// TIA Portal V19 export
FUNCTION_BLOCK "TYPIC_C301_BF_VEN"   // FB2, FBD
TITLE = TYPIC_C301_BF_VEN: Ventilatie verkeerskoker
{ S7_Optimized_Access := 'TRUE' }
AUTHOR : OCOTECH
FAMILY : Typical
NAME : C301.801
// Logisch Object Besturing: C301.801
// 
// Het doel van de BF ventilatie is de algemene opvolging, sturing en bediening van de ventilatie van een verkeerskoker.
// stored: MemoryReserve 10, SetENOAutomatically false
   VAR_INPUT
      CFG_TST_UTYD { ExternalAccessible := 'False'; ExternalVisible := 'False'; ExternalWritable := 'False'} : Time;   // Maximale transitietijd stand verandering ventilatie (transitiestatus niet bereikt)
      CFG_TST_OK_TYD { ExternalAccessible := 'False'; ExternalVisible := 'False'; ExternalWritable := 'False'} : Time;   // Stabilisatietijd voor de toestand OK (bereikt)
      CFG_ONHD_TYD { ExternalAccessible := 'False'; ExternalVisible := 'False'; ExternalWritable := 'False'} : Time;   // Waarschuwingstijd start automatische onderhoudstesten
      CFG_MAX_NOK1 { ExternalAccessible := 'False'; ExternalVisible := 'False'; ExternalWritable := 'False'} : Int;   // Maximum aantal onbestuurbare ventilatoren voor beschikbaarheidsstatus beschikbaar
      CFG_MAX_NOK2 { ExternalAccessible := 'False'; ExternalVisible := 'False'; ExternalWritable := 'False'} : Int;   // Maximum aantal onbestuurbare ventilatoren voor beschikbaarheidsstatus beperkt beschikbaar
      STU_CMD_AUT { ExternalAccessible := 'False'; ExternalVisible := 'False'; ExternalWritable := 'False'} : USInt;   // Groepscommando: schakel in automatisch
      STU_AUT_CMD { ExternalAccessible := 'False'; ExternalVisible := 'False'; ExternalWritable := 'False'} : USInt;   // Sturing ventilatie algemeen
      STU_AUT_CMD_DIR { ExternalAccessible := 'False'; ExternalVisible := 'False'; ExternalWritable := 'False'} : USInt;   // Sturing richting
      STU_AUT_VGV_BEV { ExternalAccessible := 'False'; ExternalVisible := 'False'; ExternalWritable := 'False'} : USInt;   // Vrijgave ventilator-beveiligingen onbalans en temperatuur
      STU_VGV_ONHD { ExternalAccessible := 'False'; ExternalVisible := 'False'; ExternalWritable := 'False'} : USInt;   // Vrijgave uitvoeren automatische onderhoudstesten
      STU_ALG_LCK_SIG { ExternalAccessible := 'False'; ExternalVisible := 'False'; ExternalWritable := 'False'} : USInt;   // Onderdruk alarmen
      STU_REG_CAPA { ExternalAccessible := 'False'; ExternalVisible := 'False'; ExternalWritable := 'False'} : USInt;   // Gewenste stand ventilatie bij sensorregeling (afkomstig van CF zichthandhaving)
      STU_ENE_VGV_AAN { ExternalAccessible := 'False'; ExternalVisible := 'False'; ExternalWritable := 'False'} : USInt;   // Vrijgeven of verhinderen bijschakelen energieverbruikers (verlichting / ventilatie)
      STU_ENE_MAX_AAN { ExternalAccessible := 'False'; ExternalVisible := 'False'; ExternalWritable := 'False'} : USInt;   // Maximaal toegelaten ventilatiestand
   END_VAR
   VAR_OUTPUT
      STU_CLUST { ExternalAccessible := 'False'; ExternalVisible := 'False'; ExternalWritable := 'False'} : "C301_STU_CLUST_TYPIC";   // Groepscommando met sturingen naar alle clusters van de ventilatiezone
      VAR_PWR { ExternalAccessible := 'False'; ExternalVisible := 'False'; ExternalWritable := 'False'} : Real;   // Som actueel vermogen van alle clusters
      VAR_CAPA { ExternalAccessible := 'False'; ExternalVisible := 'False'; ExternalWritable := 'False'} : USInt;   // De ingestelde ventilatiestand
      VAR_DIR { ExternalAccessible := 'False'; ExternalVisible := 'False'; ExternalWritable := 'False'} : USInt;   // De ingestelde ventilatierichting
   END_VAR
   VAR_IN_OUT
      CFG_CAPA_DIR1 : Array[1..8] of USInt;   // Omzetting ventilatiestand naar aantal ventilatoren, per cluster (zie verder), rijrichting
      CFG_CAPA_DIR2 : Array[1..8] of USInt;   // Omzetting ventilatiestand naar aantal ventilatoren, per cluster (zie verder), tegenrijrichting
      VAR_CLUST : Array[*] of "C301_VAR_CLUST_TYPIC";   // Array met alle clusters, met alle variabelen van de cluster
   END_VAR
   VAR
      BED : Struct   // Bedieningen
         ALG : Struct   // Gewenste stand
            X : "UDT_BED_ALG";
            KNOP { S7_SetPoint := 'True'} : Array[0..10] of "UDT_BED_KNOP";
         END_STRUCT;
         ALG_DIR : Struct   // Gewenste richting
            X : "UDT_BED_ALG";
            KNOP { S7_SetPoint := 'True'} : Array[0..2] of "UDT_BED_KNOP";
         END_STRUCT;
         VGV_BEV : Struct   // Vrijgave ventilator-beveiligingen onbalans en temperatuur
            X : "UDT_BED_ALG";
            KNOP { S7_SetPoint := 'True'} : Array[0..2] of "UDT_BED_KNOP";
         END_STRUCT;
         ONHD : Struct   // Uitvoeren automatische onderhoudstesten
            X : "UDT_BED_ALG";
            KNOP { S7_SetPoint := 'True'} : Array[0..1] of "UDT_BED_KNOP";
         END_STRUCT;
      END_STRUCT;
      BED_ALG { ExternalWritable := 'False'} : "TYPIC_HF_BED_ALG_KNOP";   // Gewenste stand
      BED_ALG_DIR { ExternalWritable := 'False'} : "TYPIC_HF_BED_ALG_KNOP";   // Gewenste richting
      BED_VGV_BEV { ExternalWritable := 'False'} : "TYPIC_HF_BED_ALG_KNOP";   // Vrijgave ventilator-beveiligingen onbalans en temperatuur
      BED_ONHD { ExternalWritable := 'False'} : "TYPIC_HF_BED_ALG_KNOP";   // Uitvoeren automatische onderhoudstesten
      SIG { ExternalWritable := 'False'} : Struct   // Signaleringen
         AA01 : Bool;   // Gewenste stand niet bereikt
         AA02 : Bool;   // Automatische onderhoudstesten ventilatie
         AB01 : Bool;   // Ventilatie niet beschikbaar
         AB02 : Bool;   // Ventilatie beperkt beschikbaar
      END_STRUCT;
      VAR { ExternalWritable := 'False'} : Struct   // Variabelen
         AUT_SWA : USInt;   // De stand die de ventilatie moet handhaven als de bedieningswijze is ingesteld op automatisch
         REG_CAPA : USInt;   // De stand die de ventilatie moet handhaven als de sensorregeling actief is. Deze waarde wordt bepaald door de coordinerende functie Zichthandhaving Verkeerskoker
         BMO : USInt;   // Bedieningsmode
         AUT_DIR : USInt;   // De richting die de ventilatoren op moeten blazen als de bedieningswijze is ingesteld op automatisch
         DIR_BWA : USInt;   // De werkelijke ventilatierichting
         NIV_BWA : USInt;   // Momentane ventilatieniveau (percentage)
         NIV_AAN_BWA { ExternalAccessible := 'False'; ExternalVisible := 'False'} : USInt;   // Momentaan aantal aangeschakelde ventilatoren
         NIV_AAN_SWA { ExternalAccessible := 'False'; ExternalVisible := 'False'} : USInt;   // Gewenst aantal aangeschakelde ventilatoren
         CAPA_MAX { ExternalAccessible := 'False'; ExternalVisible := 'False'} : USInt;   // Totaal aantal ventilatoren in de ventilatiezone
         CAPA_OK_BWA { ExternalAccessible := 'False'; ExternalVisible := 'False'} : USInt;   // Aantal beschikbare ventilatoren
         CAPA_BWA : USInt;   // De totaal beschikbare ventilatiecapaciteit.
         TST_BWA : USInt;   // De status van de transitie van de langsventilatie
         BSC : USInt;   // Geeft de beschikbaarheid van de langsventilatie aan
         VGV_SIG_VOP : USInt;   // TRUE = Signaleringen vrijgegeven voor verkeersoperator FALSE = Onderdrukt
         ONHD_STS : USInt;   // Status automatische onderhoudstesten
         ONHD_CLUST : USInt;   // Nummer van de cluster die onderhoudstesten dient uit te voeren
         VGV_BEV : USInt;   // Vrijgave ventilator-beveiligingen onbalans en temperatuur
         CAPA : USInt;   // De ingestelde ventilatiestand
         DIR : USInt;   // De ingestelde ventilatierichting
      END_STRUCT;
      HF_TST { ExternalAccessible := 'False'; ExternalVisible := 'False'; ExternalWritable := 'False'} : "TYPIC_HF_TST";   // Hulpfunctie transitiestatus
   END_VAR
   // // BED.ALG.KNOP[0] : Auto
   // // BED.ALG.KNOP[1] : 0 (Uit)
   // // BED.ALG.KNOP[2] : 1
   // // BED.ALG.KNOP[3] : 2
   // // BED.ALG.KNOP[4] : 3
   // // BED.ALG.KNOP[5] : 4
   // // BED.ALG.KNOP[6] : 5
   // // BED.ALG.KNOP[7] : 6
   // // BED.ALG.KNOP[8] : 7
   // // BED.ALG.KNOP[9] : 8
   // // BED.ALG.KNOP[10] : Sensorregeling
   // // BED.ALG_DIR.KNOP[0] : Auto
   // // BED.ALG_DIR.KNOP[1] : Rijrichting
   // // BED.ALG_DIR.KNOP[2] : Tegenrij
   // // BED.VGV_BEV.KNOP[0] : Auto
   // // BED.VGV_BEV.KNOP[1] : Ja
   // // BED.VGV_BEV.KNOP[2] : Onderdrukt
   // // BED.ONHD.KNOP[0] : Aan
   // // BED.ONHD.KNOP[1] : Uit
BEGIN

REGION Network 1: START
END_REGION

REGION Network 2: +++ Bedieningen +++
   // Vrijgave en verwerking van de bedieningen (centrale en lokale bediening). De bedienwaardes worden daarna in de verdere deelfunctionaliteiten gebruikt.
END_REGION

REGION Network 3: Knoppen BED_ALG(Gewenste stand)
   // Waardes en vrijge van de knoppen BED_ALG
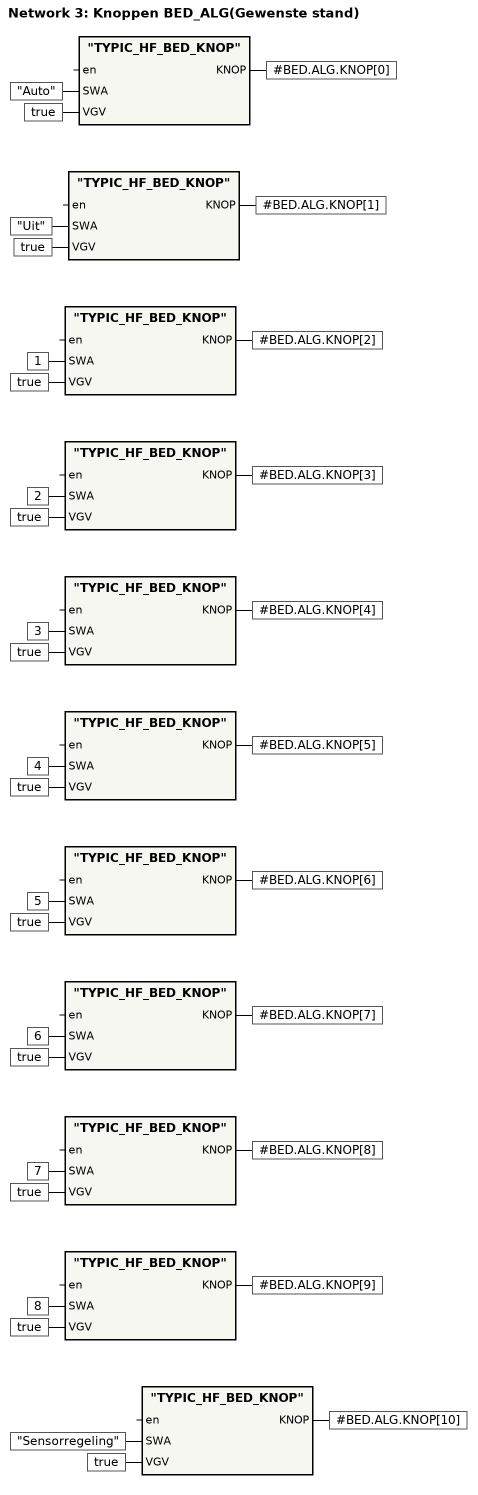
   "TYPIC_HF_BED_KNOP"(SWA := "Auto", VGV := true, KNOP => #BED.ALG.KNOP[0]);
   "TYPIC_HF_BED_KNOP"(SWA := "Uit", VGV := true, KNOP => #BED.ALG.KNOP[1]);
   "TYPIC_HF_BED_KNOP"(SWA := 1, VGV := true, KNOP => #BED.ALG.KNOP[2]);
   "TYPIC_HF_BED_KNOP"(SWA := 2, VGV := true, KNOP => #BED.ALG.KNOP[3]);
   "TYPIC_HF_BED_KNOP"(SWA := 3, VGV := true, KNOP => #BED.ALG.KNOP[4]);
   "TYPIC_HF_BED_KNOP"(SWA := 4, VGV := true, KNOP => #BED.ALG.KNOP[5]);
   "TYPIC_HF_BED_KNOP"(SWA := 5, VGV := true, KNOP => #BED.ALG.KNOP[6]);
   "TYPIC_HF_BED_KNOP"(SWA := 6, VGV := true, KNOP => #BED.ALG.KNOP[7]);
   "TYPIC_HF_BED_KNOP"(SWA := 7, VGV := true, KNOP => #BED.ALG.KNOP[8]);
   "TYPIC_HF_BED_KNOP"(SWA := 8, VGV := true, KNOP => #BED.ALG.KNOP[9]);
   "TYPIC_HF_BED_KNOP"(SWA := "Sensorregeling", VGV := true, KNOP => #BED.ALG.KNOP[10]);
END_REGION

REGION Network 4: BED_ALG(Gewenste stand)
   // Verwerking BED_ALG
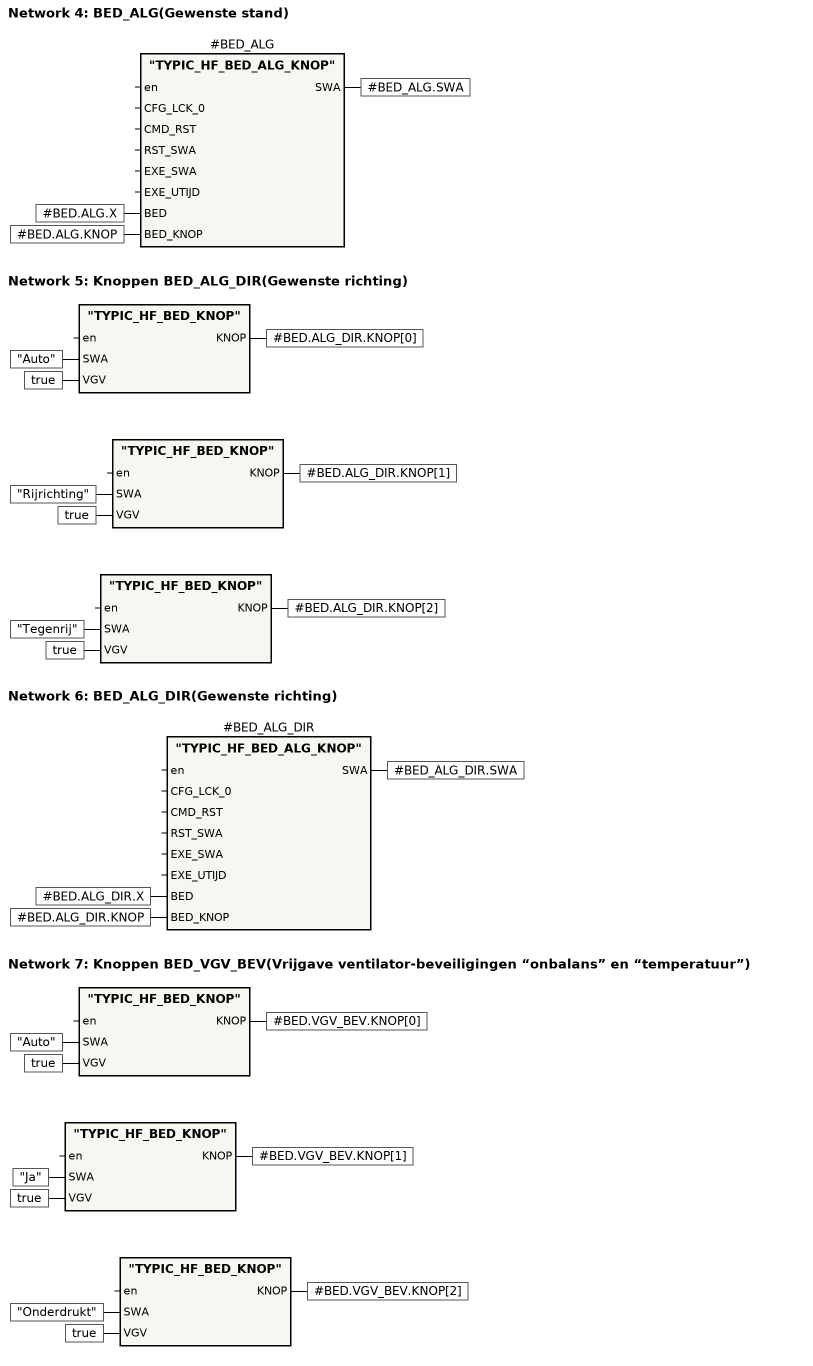
   #BED_ALG(BED := #BED.ALG.X, BED_KNOP := #BED.ALG.KNOP, SWA => #BED_ALG.SWA);   // "TYPIC_HF_BED_ALG_KNOP"
END_REGION

REGION Network 5: Knoppen BED_ALG_DIR(Gewenste richting)
   // Waardes en vrijge van de knoppen BED_ALG_DIR
   "TYPIC_HF_BED_KNOP"(SWA := "Auto", VGV := true, KNOP => #BED.ALG_DIR.KNOP[0]);
   "TYPIC_HF_BED_KNOP"(SWA := "Rijrichting", VGV := true, KNOP => #BED.ALG_DIR.KNOP[1]);
   "TYPIC_HF_BED_KNOP"(SWA := "Tegenrij", VGV := true, KNOP => #BED.ALG_DIR.KNOP[2]);
END_REGION

REGION Network 6: BED_ALG_DIR(Gewenste richting)
   // Verwerking BED_ALG_DIR
   #BED_ALG_DIR(BED := #BED.ALG_DIR.X, BED_KNOP := #BED.ALG_DIR.KNOP, SWA => #BED_ALG_DIR.SWA);   // "TYPIC_HF_BED_ALG_KNOP"
END_REGION

REGION Network 7: Knoppen BED_VGV_BEV(Vrijgave ventilator-beveiligingen “onbalans” en “temperatuur”)
   // Waardes en vrijge van de knoppen BED_VGV_BEV
   "TYPIC_HF_BED_KNOP"(SWA := "Auto", VGV := true, KNOP => #BED.VGV_BEV.KNOP[0]);
   "TYPIC_HF_BED_KNOP"(SWA := "Ja", VGV := true, KNOP => #BED.VGV_BEV.KNOP[1]);
   "TYPIC_HF_BED_KNOP"(SWA := "Onderdrukt", VGV := true, KNOP => #BED.VGV_BEV.KNOP[2]);
END_REGION

REGION Network 8: BED_VGV_BEV(Vrijgave ventilator-beveiligingen “onbalans” en “temperatuur”)
   // Verwerking BED_VGV_BEV
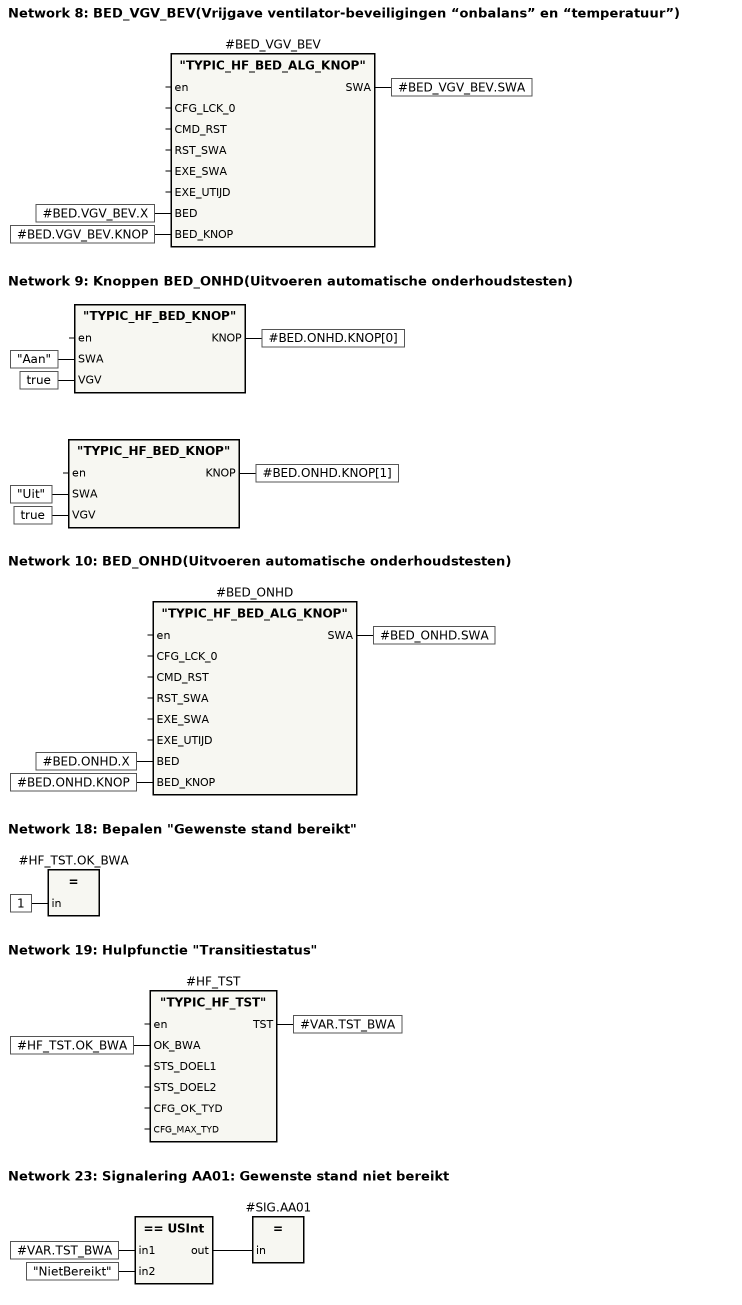
   #BED_VGV_BEV(BED := #BED.VGV_BEV.X, BED_KNOP := #BED.VGV_BEV.KNOP, SWA => #BED_VGV_BEV.SWA);   // "TYPIC_HF_BED_ALG_KNOP"
END_REGION

REGION Network 9: Knoppen BED_ONHD(Uitvoeren automatische onderhoudstesten)
   // Waardes en vrijge van de knoppen BED_ONHD
   "TYPIC_HF_BED_KNOP"(SWA := "Aan", VGV := true, KNOP => #BED.ONHD.KNOP[0]);
   "TYPIC_HF_BED_KNOP"(SWA := "Uit", VGV := true, KNOP => #BED.ONHD.KNOP[1]);
END_REGION

REGION Network 10: BED_ONHD(Uitvoeren automatische onderhoudstesten)
   // Verwerking BED_ONHD
   #BED_ONHD(BED := #BED.ONHD.X, BED_KNOP := #BED.ONHD.KNOP, SWA => #BED_ONHD.SWA);   // "TYPIC_HF_BED_ALG_KNOP"
END_REGION

REGION Network 11: +++ Bepalen bedieningsmode +++
   // Bedieningsmode (Auto / Manueel ) bepalen.
END_REGION

REGION Network 12: +++ Bepalen gewenste capaciteitsinstelling +++
   // Bepalen van de gewenste stand (0..8).
END_REGION

REGION Network 13: +++ Bepalen gewenste ventilatierichting +++
   // Bepalen van de gewenste draairichting (Rijrichting / Tegenrij).
END_REGION

REGION Network 14: +++ Bepalen vrijgave ventilatorbeveiligingen +++
   // Bepalen vrijgave of onderdrukken van de ventilatorbeveiligingen onbalans en temperatuur.
END_REGION

REGION Network 15: +++ Bepalen werkelijke ventilatierichting +++
   // Bepalen van de werkelijke ventilatierichting (Rijrichting / Tegenrij / Onbepaald) aan de hand van de ventilatierichtingen van de ventilatieclusters.
END_REGION

REGION Network 16: +++ Berekeningen +++
   // Verscheidene berekeningen die nodig zijn voor de functionele werking of info voor weergave via de centrale en lokale bediening, zoals het momentane ventilatieniveau, aantal beschikbare ventilatoren, beschikbare capaciteit, actueel vermogen ventilatiezone.
END_REGION

REGION Network 17: +++ Bepalen transitiestatus +++
   // Transitiestatus (bereikt / niet bereikt / in transitie) bepalen.
END_REGION

REGION Network 18: Bepalen "Gewenste stand bereikt"
   // Bepalen of de actuele stand in overeenstemming is met de gewenste stand
   #HF_TST.OK_BWA := 1;
END_REGION

REGION Network 19: Hulpfunctie "Transitiestatus"
   // De transitiestatus geeft de relatie tussen een gewenste stand (van een functionaliteit) en de actuele stand aan.
   #HF_TST(OK_BWA := #HF_TST.OK_BWA, TST => #VAR.TST_BWA);   // "TYPIC_HF_TST"
END_REGION

REGION Network 20: +++ Bepalen beschikbaarheidsstatus +++
   // Beschikbaarheidsstatus (beschikbaar / beperkt beschikbaar / niet beschikbaar) bepalen.
END_REGION

REGION Network 21 (SCL): Beschikbaarheidsstatus bepalen
   IF 
       //voorwaarden "Niet beschikbaar"
       TRUE
   THEN
       //Beschikbaarheidsstatus = Niet Beschikbaar
       #VAR.BSC:= "NietBeschikbaar";
   ELSIF
       //voorwaarden "Beperkt beschikbaar"
       TRUE
   THEN
       //Beschikbaarheidsstatus = Beperkt Beschikbaar
       #VAR.BSC:= "Beperkt";
   ELSE
       //Beschikbaarheidsstatus = Beschikbaar
       #VAR.BSC:= "Beschikbaar";
   END_IF;
END_REGION

REGION Network 22: +++ Signaleringen +++
   // Aanmaken signaleringen.
END_REGION

REGION Network 23: Signalering AA01: Gewenste stand niet bereikt
   #SIG.AA01 := #VAR.TST_BWA = "NietBereikt";
END_REGION

REGION Network 24: Signalering AB01 : Niet Beschikbaar
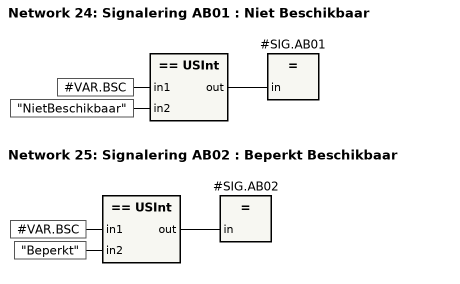
   #SIG.AB01 := #VAR.BSC = "NietBeschikbaar";
END_REGION

REGION Network 25: Signalering AB02 : Beperkt Beschikbaar
   #SIG.AB02 := #VAR.BSC = "Beperkt";
END_REGION

REGION Network 26: +++ Automatische onderhoudstesten +++
   // Functionaliteit waarbij iedere ventilator een voor een aangestuurd wordt ter controle van de goede werking van iedere ventilator.
END_REGION

REGION Network 27: +++ Sturingen +++
   // Uitgeven van sturingen naar de ventilatieclusters.
END_REGION

REGION Network 28: EINDE
   // Variabelen van intern scada rakvlak naar outputs copieren
END_REGION
END_FUNCTION_BLOCK
